// TIA Portal V20 export
// export: Created 2025-12-01T14:57:32.0244109Z, ExportSetting None, DisplayName Totally Integrated Automation Portal, DisplayVersion V20 Update 3, DisplayName TIA Portal Openness, DisplayVersion V20 Update 3, DisplayName TIA Portal Version Control Interface, DisplayVersion V20 Update 3, DisplayName STEP 7 Professional, DisplayVersion V20 Update 3, DisplayName STEP 7 Safety, DisplayVersion V20 Update 2, DisplayName WinCC Basic/Comfort/Advanced, DisplayVersion V20 Update 3, DisplayName WinCC Professional, DisplayVersion V20 Update 3, DisplayName WinCC Unified, DisplayVersion V20 Update 3
DATA_BLOCK "DB771_HMI_VTD"   // DB771
{ S7_Optimized_Access := 'FALSE' }
// stored: AutoNumber false
   VAR
      Dispositivo : Array[0..15] of Struct
         Estado_Variador : Struct
            "Estatus variador" { S7_SetPoint := 'True'} : "i950 Estatus variador";   // Word que informa del estado del dispositivo
            "Palabra de control" : "i950 Palabra de Control";   // Word que controla la activación del dispositvo
            "Código de error" : DInt;   // Código proporcionado por Lenze para diagnosticar el fallo
         END_STRUCT;
         Position_Actual : DInt;
         Position_Destino : DInt;
         Mov_Manual : Struct
            MesaHorquilla : UInt;
            MesaDestino : UInt;
            Remoto_OK : Bool;
            Bussy : Bool;
            Free_2 : Bool;
            Free_3 : Bool;
            Free_4 : Bool;
            Free_5 : Bool;
            Free_6 : Bool;
            Free_7 : Bool;
            Avance : Bool;
            Retroceso : Bool;
            Enviar_Orden : Bool;
            Confirmar_Orden : Bool;
            Free1_4 : Bool;
            Free1_5 : Bool;
            Free1_6 : Bool;
            Free1_7 : Bool;
         END_STRUCT;
         EstadoVTD { S7_SetPoint := 'True'} : "EstadoZona";
         Free_Word : Word;
      END_STRUCT;
   END_VAR
BEGIN
END_DATA_BLOCK
